(* IEC 61131-3 sources: mect_apps/TP1043_TCP/ModbusTCPclient_CFG/Output, 1 file *)

(* ---- Resource1.gvl ---- *)
VAR_GLOBAL
DigitalOutput_1 AT %MW0.5380:INT;
DigitalOutput_2 AT %MW0.5384:INT;
DigitalInput_3 AT %MW0.5388:INT;
DigitalInput_4 AT %MW0.5392:INT;
TimeValue AT %MD0.5396:REAL;
TimeValueMin AT %MD0.5400:REAL;
TimeValueMax AT %MD0.5404:REAL;
AnalogInput_1 AT %MW0.5408:INT;
AnalogInput_2 AT %MW0.5412:INT;
END_VAR
